DATA_BLOCK "DB_KeyenceCheckerIV3"
VAR
  aDev : Array[1..4] of "ST_KeyenceCheckerIV3";
END_VAR
BEGIN
END_DATA_BLOCK
